FUNCTION alg_a_DledQ2 : BOOL
VAR_INPUT
	state: STATE;
END_VAR

alg_a_DledQ2 := FALSE;

END_FUNCTION

(* stored: Version 1.1.0.1, ProductVersion 3.1.4022.18
   POU alg_a_DledQ2: Id {a0439a55-6024-43fc-97cf-a117b05af963}, SpecialFunc None *)
